TYPE ST_System_HOWW_Stellwert :
STRUCT
	Anford_Stellventil		: BOOL;
	Anford_Pumpe		: BOOL;
	Freigabe_Anlage		: BOOL;
END_STRUCT
END_TYPE

(* stored: Version 1.1.0.1, ProductVersion 3.1.4024.9
   DUT ST_System_HOWW_Stellwert: Id {f65493a4-9872-4baf-88a0-80857d669f60} *)
